// TIA Portal V17 export
// export: Created 2024-09-03T21:55:02.5108022Z, ExportSetting WithDefaults, DisplayName Totally Integrated Automation Portal, DisplayVersion V17 Update 7, DisplayName TIA Portal Openness, DisplayVersion V17 Update 7, DisplayName TIA Portal Version Control Interface, DisplayVersion V17, DisplayName SINAMICS Startdrive Advanced, DisplayVersion V17 SP2, DisplayName SINAMICS Startdrive G110M, G120, G120C, G120D, G120P, G115D, DisplayVersion V17 SP2, DisplayName SINAMICS Startdrive G130, G150, S120, S150, SINAMICS MV, S210, DisplayVersion V17 SP2, DisplayName STEP 7 Professional, DisplayVersion V17 Update 7, DisplayName STEP 7 Safety, DisplayVersion V17 Update 6, DisplayName WinCC Advanced / Unified PC, DisplayVersion V17 Update 7
VAR_GLOBAL   // PLC tag table "hmi"
   iBtnBasicPosition AT %I125.3 : Bool;
   qBasicPosition AT %Q125.1 : Bool;
   qResetAlarm AT %Q125.2 : Bool;
   iBtnResetAlarm AT %I125.4 : Bool;
   iBtnStart AT %I125.2 : Bool;
   qStart AT %Q125.0 : Bool;
   iBtnStartAuto AT %I125.7 : Bool;
   qAuto AT %Q125.3 : Bool;
   qManual AT %Q125.4 : Bool;
   iManual AT %I125.5 : Bool;
   iAuto AT %I125.6 : Bool;
END_VAR
